// Block: PPrgArchive17

DATA_BLOCK PPrgArchive17
VERSION : 0.1
   NON_RETAIN
   VAR
      PRG : Array[1601..1700] of PPrg_Data;
   END_VAR

BEGIN
   // No initialization required
END_DATA_BLOCK
